// Mitsubishi GX Works2 project: Group15   PLC: FX3G

// global labels: Global1
VAR_GLOBAL
  StartSwitch AT X007 : BOOL;
  BreakSwitch AT X011 : BOOL;
  WorkDayLight AT Y007 : BOOL;
  Start_cooking AT X001 : BOOL;
  Analog_input_1 AT D8280 : INT;
  Save_analog_input_1 AT D8200 : REAL;
  Cooking_input_indicator AT M0 : BOOL;
END_VAR
VAR_GLOBAL CONSTANT
  Const_5 : REAL := 5;
END_VAR
VAR_GLOBAL
  Save_yeast AT D2000 : REAL;
  Save_hops AT D3000 : REAL;
  Save_malt AT D4000 : REAL;
END_VAR
VAR_GLOBAL CONSTANT
  lagger_yeast : REAL := 150.0;
  lagger_malt : REAL := 12.0;
  lagger_hops : REAL := 60.0;
  Const_6 : REAL := 6;
  filzner_yeast : REAL := 120.0;
  filzner_malt : REAL := 6.0;
  filzner_hops : REAL := 54.0;
END_VAR
VAR_GLOBAL
  Cooking_light AT Y001 : BOOL;
  Cooking_timer_TC_1 AT TC1 : BOOL;
END_VAR
VAR_GLOBAL CONSTANT
  Timer_value_4_sec : INT := 40;
END_VAR
VAR_GLOBAL
  End_cooking_TS_1 AT TS1 : BOOL;
  Analog_input_under_5 AT M1 : BOOL;
  Analog_input_above_6 AT M2 : BOOL;
END_VAR
VAR_GLOBAL CONSTANT
  Convert : REAL := 400;
END_VAR
VAR_GLOBAL
  Ready_to_cook_lagger AT M3 : BOOL;
  Ready_to_cook_filzner AT M4 : BOOL;
  Start_fizzing AT X005 : BOOL;
  Cooking_container AT D5000 : REAL;
END_VAR
VAR_GLOBAL CONSTANT
  Cooking_sum_lagger : REAL := 222.0;
  Cooking_sum_filzner : REAL := 180.0;
END_VAR
VAR_GLOBAL
  Fizzing_container AT D6000 : REAL;
  Fizzing_container_full AT M5 : BOOL;
  Fizzing_in_process AT M6 : BOOL;
  Fizzing_timer_lagger_TC_2 AT TC2 : BOOL;
END_VAR
VAR_GLOBAL CONSTANT
  Timer_value_3_sec : INT := 30;
  Fizzing_timer_filzner_TC_3 : BOOL;
END_VAR
VAR_GLOBAL
  Start_packing AT X002 : BOOL;
  End_fizzing_lagger AT TS2 : BOOL;
  End_fizzing_TS_3 AT TS3 : BOOL;
  Fizzing_light_1 AT Y003 : BOOL;
  Flicker_light_Y3_timer AT TC4 : BOOL;
END_VAR
VAR_GLOBAL CONSTANT
  Timer_value_075_sec : REAL := 7.5;
END_VAR
VAR_GLOBAL
  End_one_flicker_Y3 AT TS4 : BOOL;
  Fizzing_light_2 AT Y004 : BOOL;
  Flicker_light_Y4_timer AT TC5 : BOOL;
  End_one_flicker_Y4 AT TS5 : BOOL;
END_VAR
VAR_GLOBAL CONSTANT
  Timer_value_07_sec : INT := 5;
END_VAR
VAR_GLOBAL
  Packing_bottle AT X000 : BOOL;
  Packing_light AT Y002 : BOOL;
  Counting_6_pack AT CC1 : BOOL;
END_VAR
VAR_GLOBAL CONSTANT
  Val_5 : INT := 5;
END_VAR
VAR_GLOBAL
  End_packing_CS_1 AT CS1 : BOOL;
  Storage_container AT D7000 : REAL;
END_VAR
VAR_GLOBAL CONSTANT
  One_package : REAL := 0.1;
END_VAR
VAR_GLOBAL
  Analog_output AT D8282 : INT;
END_VAR
VAR_GLOBAL CONSTANT
  Six_pack : REAL := 1.0;
END_VAR
VAR_GLOBAL
  enough_materials_for_workday AT M7 : BOOL;
  Yeast_input AT D2500 : REAL;
  Malt_input AT D4500 : REAL;
  Hops_input AT D3500 : REAL;
END_VAR
VAR_GLOBAL CONSTANT
  Yeast_min : REAL := 120.0;
  Hops_min : REAL := 54.0;
  Malt_min : REAL := 6.0;
  Enough_yeast_for_lagger : REAL := 150.0;
  Enough_hops_for_lagger : REAL := 60.0;
  Enough_malt_for_lagger : REAL := 12.0;
  Valid_to_analog_output : REAL := 10.0;
  Converting_to_analog_output : REAL := 40;
  reset_constant_word : INT;
  reset_constant_float : REAL;
END_VAR

// task Task_01 (event TRUE, interval 0, priority 31): POU_01

PROGRAM POU_01
(* structured ladder/FBD written out as ST: instructions are called as NAME(EN, inputs, outputs); _pN, _eN, _tN stand for wires *)
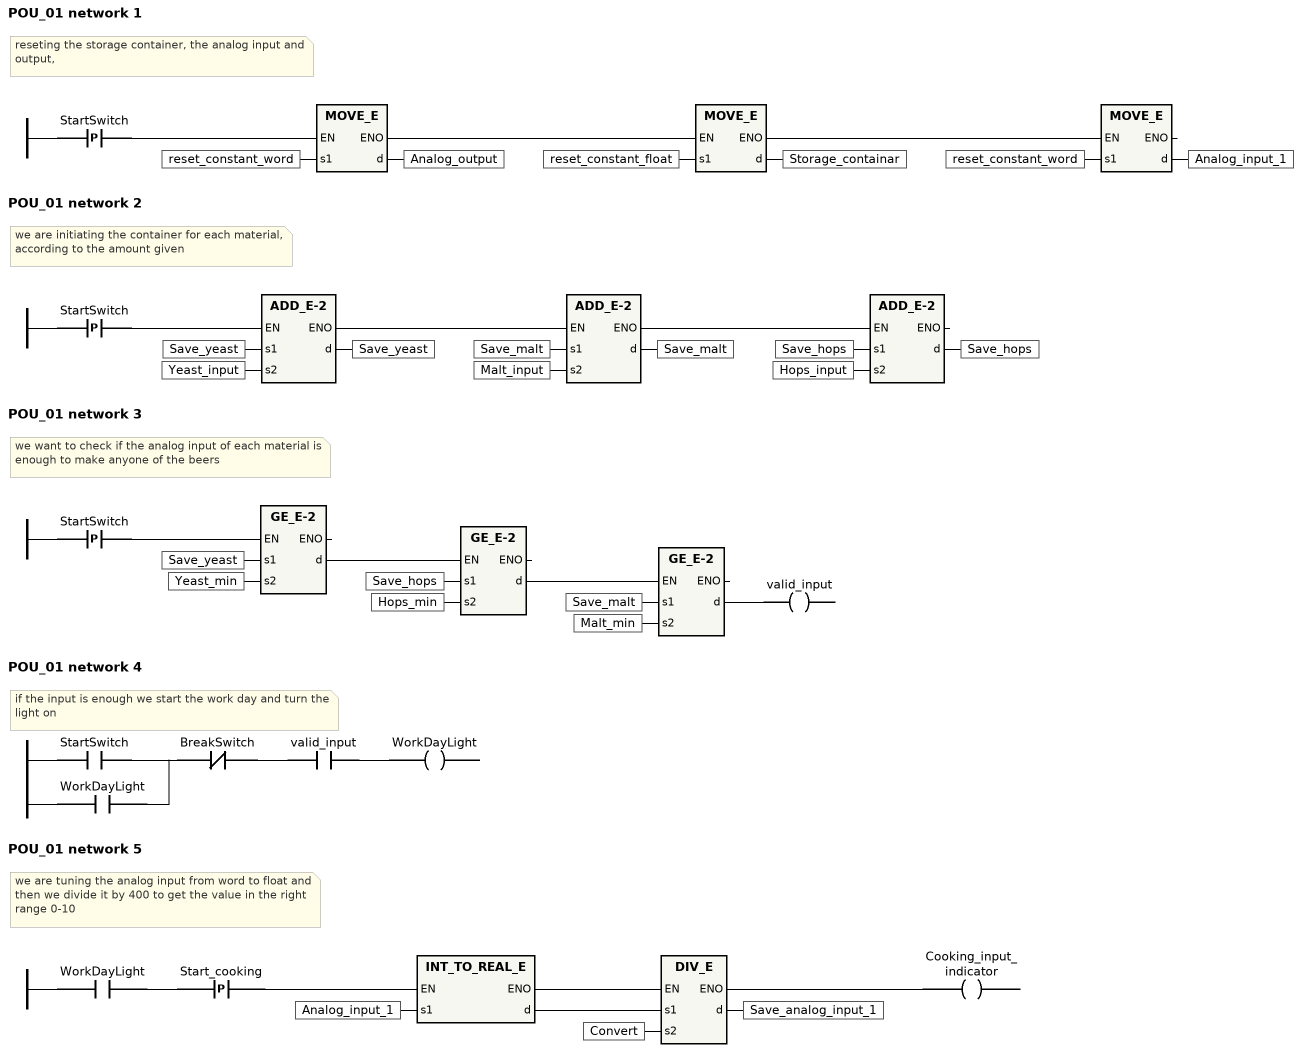
(* network 1 *)
(* reseting the storage container, the analog input and output, *)
_e1 := MOVE_E(LDP(TRUE, StartSwitch), reset_constant_word, Analog_output);
_e2 := MOVE_E(_e1, reset_constant_float, Storage_containar);
MOVE_E(_e2, reset_constant_word, Analog_input_1);
(* network 2 *)
(* we are initiating the container for each material, according to the amount given *)
_e1 := ADD_E(LDP(TRUE, StartSwitch), Save_yeast, Yeast_input, Save_yeast);
_e2 := ADD_E(_e1, Save_malt, Malt_input, Save_malt);
ADD_E(_e2, Save_hops, Hops_input, Save_hops);
(* network 3 *)
(* we want to check if the analog input of each material is enough to make anyone of the beers *)
GE_E(LDP(TRUE, StartSwitch), Save_yeast, Yeast_min, _t1);
GE_E(_t1, Save_hops, Hops_min, _t2);
GE_E(_t2, Save_malt, Malt_min, _t3);
valid_input := _t3;
(* network 4 *)
(* if the input is enough we start the work day and turn the light on *)
WorkDayLight := ((StartSwitch OR WorkDayLight) AND NOT BreakSwitch) AND valid_input;
(* network 5 *)
(* we are tuning the analog input from word to float and then we divide it by 400 to get the value in the right range 0-10 *)
_e2 := INT_TO_REAL_E(WorkDayLight AND LDP(TRUE, Start_cooking), Analog_input_1, _t1);
_e3 := DIV_E(_e2, _t1, Convert, Save_analog_input_1);
Cooking_input_indicator := _e3;
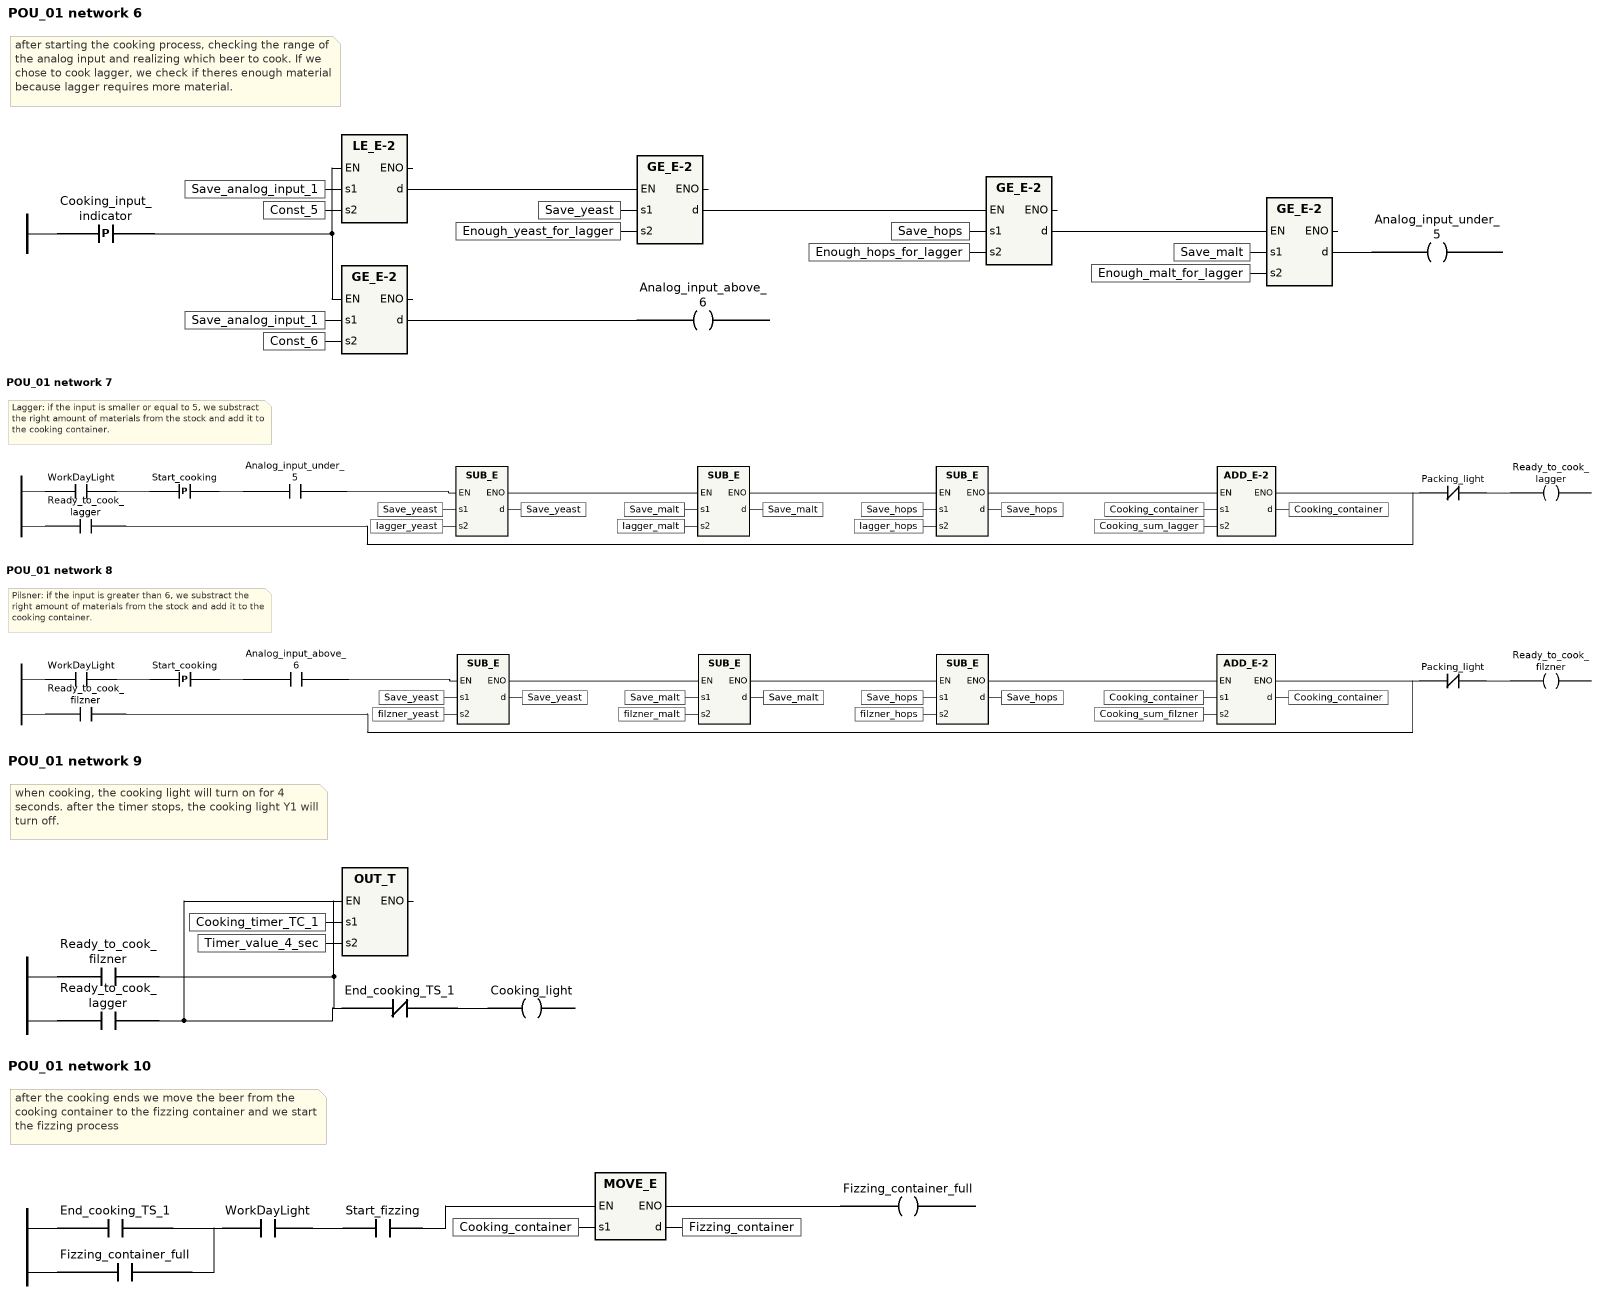
(* network 6 *)
(* after starting the cooking process, checking the range of the analog input and realizing which beer to cook. If we chose to cook lagger, we check if theres enough material because lagger requires more material. *)
_p1 := LDP(TRUE, Cooking_input_indicator);
LE_E(_p1, Save_analog_input_1, Const_5, _t2);
GE_E(_t2, Save_yeast, Enough_yeast_for_lagger, _t3);
GE_E(_t3, Save_hops, Enough_hops_for_lagger, _t4);
GE_E(_t4, Save_malt, Enough_malt_for_lagger, _t5);
Analog_input_under_5 := _t5;
GE_E(_p1, Save_analog_input_1, Const_6, _t6);
Analog_input_above_6 := _t6;
(* network 7 *)
(* Lagger: if the input is smaller or equal to 5, we substract the right amount of materials from the stock and add it to the cooking container. *)
_e1 := SUB_E(WorkDayLight AND LDP(TRUE, Start_cooking) AND Analog_input_under_5, Save_yeast, lagger_yeast, Save_yeast);
_e2 := SUB_E(_e1, Save_malt, lagger_malt, Save_malt);
_e3 := SUB_E(_e2, Save_hops, lagger_hops, Save_hops);
_e4 := ADD_E(_e3, Cooking_container, Cooking_sum_lagger, Cooking_container);
Ready_to_cook_lagger := (_e4 OR Ready_to_cook_lagger) AND NOT Packing_light;
(* network 8 *)
(* Pilsner: if the input is greater than 6, we substract the right amount of materials from the stock and add it to the cooking container. *)
_e1 := SUB_E(WorkDayLight AND LDP(TRUE, Start_cooking) AND Analog_input_above_6, Save_yeast, filzner_yeast, Save_yeast);
_e2 := SUB_E(_e1, Save_malt, filzner_malt, Save_malt);
_e3 := SUB_E(_e2, Save_hops, filzner_hops, Save_hops);
_e4 := ADD_E(_e3, Cooking_container, Cooking_sum_filzner, Cooking_container);
Ready_to_cook_filzner := (_e4 OR Ready_to_cook_filzner) AND NOT Packing_light;
(* network 9 *)
(* when cooking, the cooking light will turn on for 4 seconds. after the timer stops, the cooking light Y1 will turn off. *)
_p1 := Ready_to_cook_filzner OR Ready_to_cook_lagger;
OUT_T(_p1, Cooking_timer_TC_1, Timer_value_4_sec);
Cooking_light := _p1 AND NOT End_cooking_TS_1;
(* network 10 *)
(* after the cooking ends we move the beer from the cooking container to the fizzing container and we start the fizzing process *)
_e1 := MOVE_E(((End_cooking_TS_1 OR Fizzing_container_full) AND WorkDayLight) AND Start_fizzing, Cooking_container, Fizzing_container);
Fizzing_container_full := _e1;
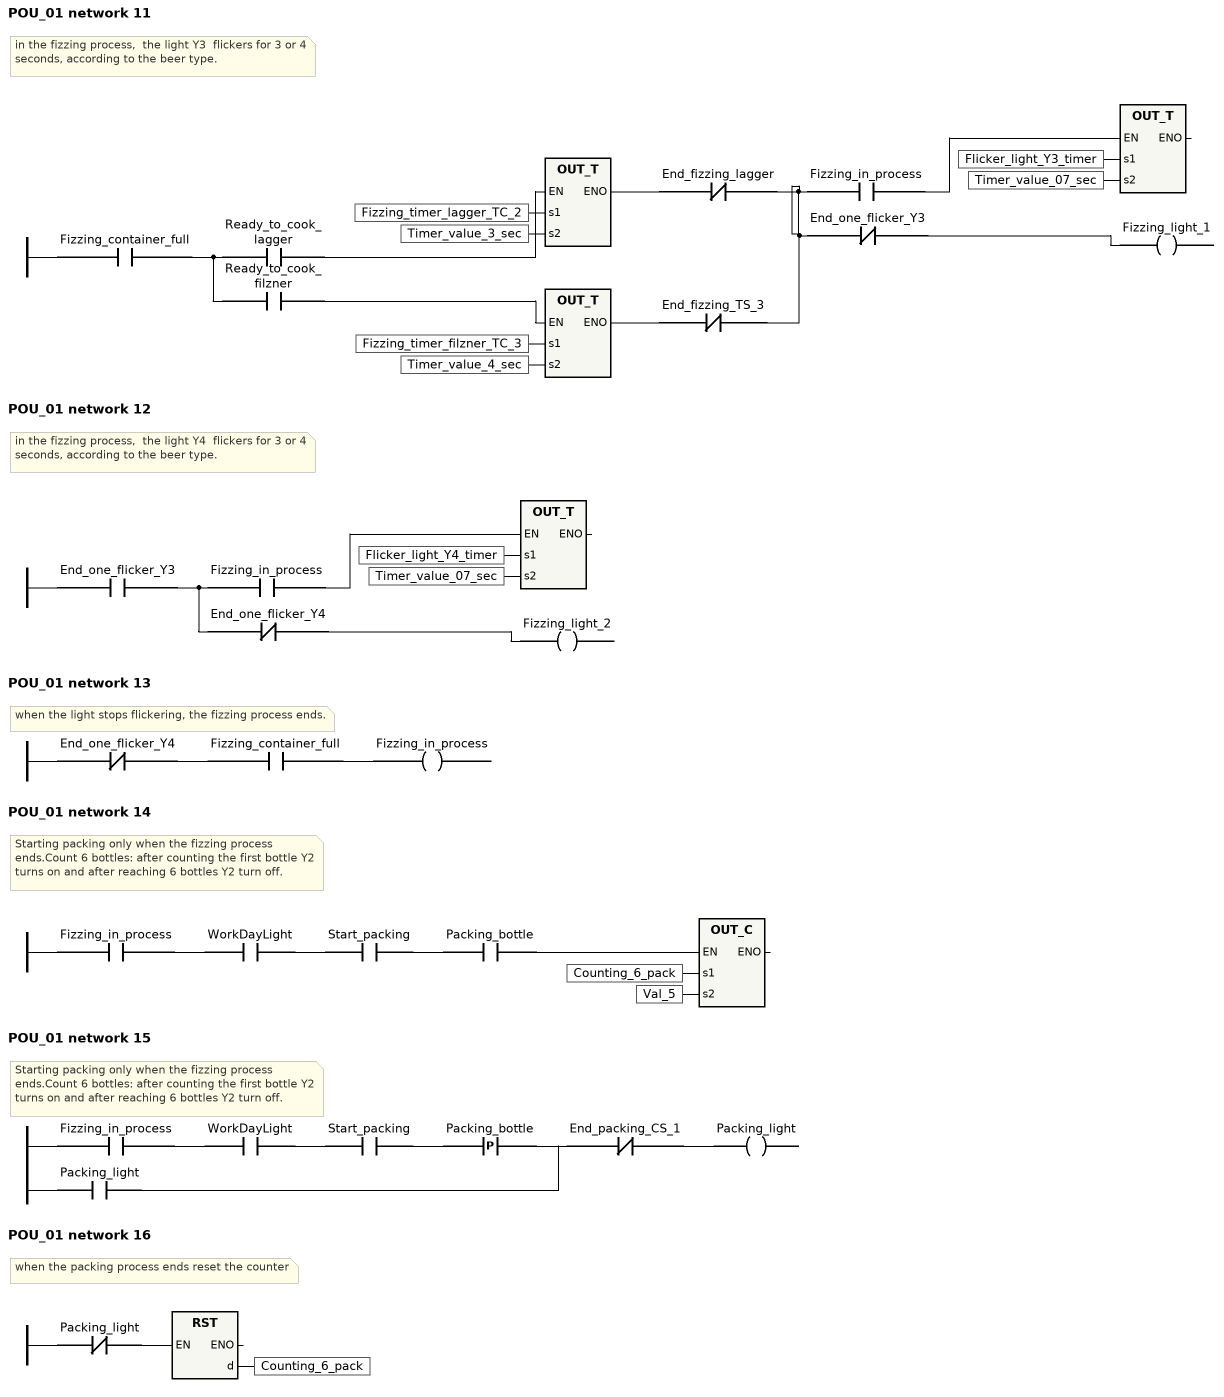
(* network 11 *)
(* in the fizzing process,  the light Y3  flickers for 3 or 4 seconds, according to the beer type. *)
_e1 := OUT_T(Fizzing_container_full AND Ready_to_cook_lagger, Fizzing_timer_lagger_TC_2, Timer_value_3_sec);
_e2 := OUT_T(Fizzing_container_full AND Ready_to_cook_filzner, Fizzing_timer_filzner_TC_3, Timer_value_4_sec);
_p3 := (_e1 AND NOT End_fizzing_lagger) OR (_e2 AND NOT End_fizzing_TS_3);
OUT_T(_p3 AND Fizzing_in_process, Flicker_light_Y3_timer, Timer_value_07_sec);
Fizzing_light_1 := _p3 AND NOT End_one_flicker_Y3;
(* network 12 *)
(* in the fizzing process,  the light Y4  flickers for 3 or 4 seconds, according to the beer type. *)
OUT_T(End_one_flicker_Y3 AND Fizzing_in_process, Flicker_light_Y4_timer, Timer_value_07_sec);
Fizzing_light_2 := End_one_flicker_Y3 AND NOT End_one_flicker_Y4;
(* network 13 *)
(* when the light stops flickering, the fizzing process ends. *)
Fizzing_in_process := NOT End_one_flicker_Y4 AND Fizzing_container_full;
(* network 14 *)
(* Starting packing only when the fizzing process ends.Count 6 bottles: after counting the first bottle Y2 turns on and after reaching 6 bottles Y2 turn off. *)
OUT_C(Fizzing_in_process AND WorkDayLight AND Start_packing AND Packing_bottle, Counting_6_pack, Val_5);
(* network 15 *)
(* Starting packing only when the fizzing process ends.Count 6 bottles: after counting the first bottle Y2 turns on and after reaching 6 bottles Y2 turn off. *)
Packing_light := ((Fizzing_in_process AND WorkDayLight AND Start_packing AND LDP(TRUE, Packing_bottle)) OR Packing_light) AND NOT End_packing_CS_1;
(* network 16 *)
(* when the packing process ends reset the counter *)
RST(NOT Packing_light, Counting_6_pack);
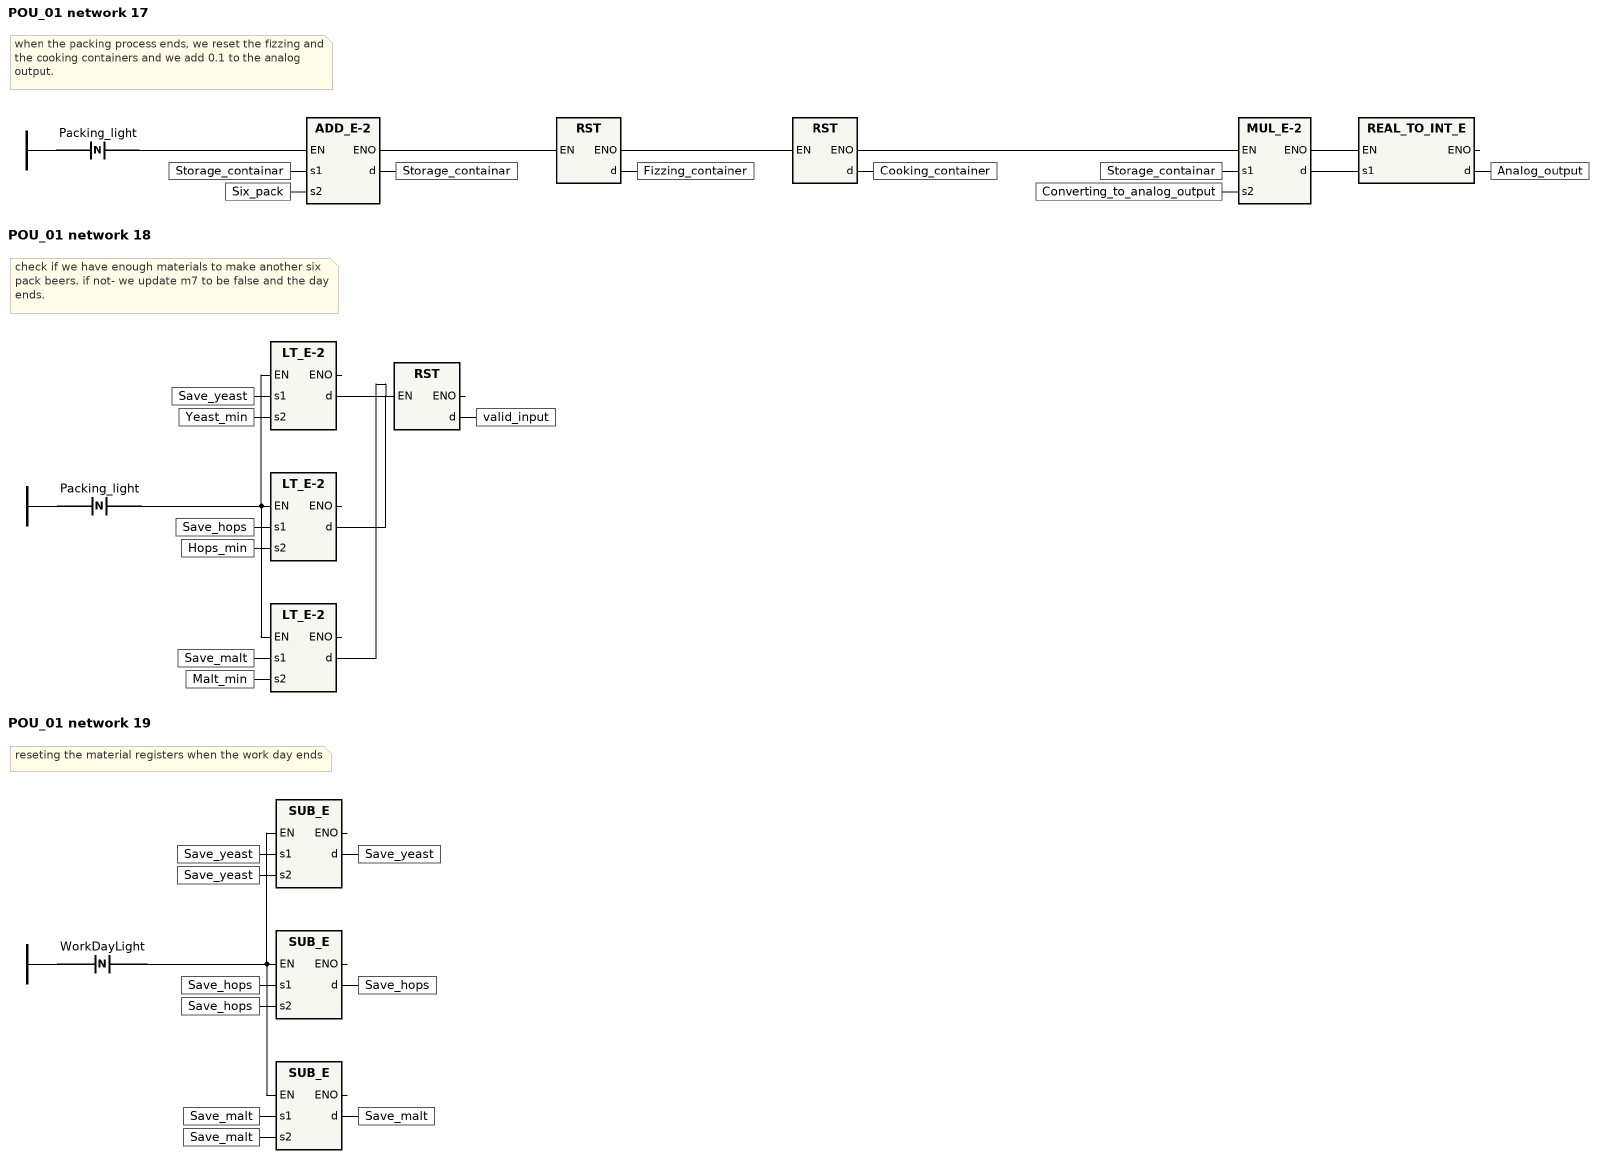
(* network 17 *)
(* when the packing process ends, we reset the fizzing and the cooking containers and we add 0.1 to the analog output. *)
_e1 := ADD_E(LDF(TRUE, Packing_light), Storage_containar, Six_pack, Storage_containar);
_e2 := RST(_e1, Fizzing_container);
_e3 := RST(_e2, Cooking_container);
_e5 := MUL_E(_e3, Storage_containar, Converting_to_analog_output, _t4);
REAL_TO_INT_E(_e5, _t4, Analog_output);
(* network 18 *)
(* check if we have enough materials to make another six pack beers. if not- we update m7 to be false and the day ends. *)
_p1 := LDF(TRUE, Packing_light);
LT_E(_p1, Save_yeast, Yeast_min, _t2);
LT_E(_p1, Save_hops, Hops_min, _t3);
LT_E(_p1, Save_malt, Malt_min, _t4);
RST(_t2 OR _t3 OR _t4, valid_input);
(* network 19 *)
(* reseting the material registers when the work day ends *)
_p1 := LDF(TRUE, WorkDayLight);
SUB_E(_p1, Save_yeast, Save_yeast, Save_yeast);
SUB_E(_p1, Save_hops, Save_hops, Save_hops);
SUB_E(_p1, Save_malt, Save_malt, Save_malt);
END_PROGRAM
